Staubli VAL3: wZone.pgx

public program wZone(tool x_tTool, point x_pPoint, frame x_fFrame, num x_Dx, num x_Dy, num x_Dz, dio& x_dOut)
begin

  //set x_dOut to false if x_tTool is inside a box defined as:

  //x_pPoint.trsf.x + x_Dx/2 > here(x_tTool, x_fFrame).x > x_pPoint.trsf.x - x_Dx/2
  //x_pPoint.trsf.y + x_Dy/2 > here(x_tTool, x_fFrame).y > x_pPoint.trsf.y - x_Dy/2
  //x_pPoint.trsf.z + x_Dz/2 > here(x_tTool, x_fFrame).z > x_pPoint.trsf.z - x_Dz/2

  if taskStatus("wZone_"+toString("",nWzoneCount))==-1
    taskCreate "wZone_"+toString("",nWzoneCount),15,exeWzone(x_tTool,x_pPoint,x_fFrame,x_Dx,x_Dy,x_Dz,x_dOut)
    nWzoneCount=nWzoneCount+1
    if nWzoneCount>nMaxTask
      nWzoneCount=0
    endIf
  else
    logMsg("libSignals/wZone->can't create the task")
  endIf


end
